FUNCTION_BLOCK FB_TofOnRtrig		// Monitors a signal (R_TRIG) and creates a TOF
VAR_INPUT
	iBool:		BOOL;	// Signal to be monitored
	iTime:		TIME;	// TOF time
END_VAR
VAR_OUTPUT
	oBool: 		BOOL;	// Set TRUE for iTime on a rising edge of iBool
END_VAR
VAR
	rtrig:		R_TRIG;
	tof:		TOF;
END_VAR

rtrig(CLK := iBool);
tof(IN := rtrig.Q, PT := iTime, Q => oBool);

END_FUNCTION_BLOCK

(* stored: Version 1.1.0.1, ProductVersion 3.1.4026.18
   POU FB_TofOnRtrig: Id {46917ec6-a9c5-40a9-b661-1b33bb463d2b}, SpecialFunc None *)
